// TIA Portal V20 export
// export: Created 2026-07-10T11:12:27.4069483Z, ExportSetting WithDefaults, DisplayName Totally Integrated Automation Portal, DisplayVersion V20, DisplayName TIA Portal Openness, DisplayVersion V20, DisplayName TIA Portal Version Control Interface, DisplayVersion V20, DisplayName STEP 7 Professional, DisplayVersion V20, DisplayName STEP 7 Safety, DisplayVersion V20, DisplayName WinCC Basic/Comfort/Advanced, DisplayVersion V20, DisplayName WinCC Unified, DisplayVersion V20
DATA_BLOCK "Inputs_DB"   // DB5
VERSION : 0.1
// stored: AutoNumber true, DBAccessibleFromOPCUA true, InstanceOfName Inputs, InstanceOfType FB
"Inputs"
   // VAR
   //    AIHandlers { S7_SetPoint := 'True'} : Array[0..5] of "AIHandler";
   //    WeightHandlers { S7_SetPoint := 'True'} : Array[0..1] of "WeightHandler";
   //    ErrorRCV1 { S7_SetPoint := 'True'} : Bool := TRUE;
   //    ErrorRCV2 { S7_SetPoint := 'True'} : Bool := TRUE;
   // END_VAR
BEGIN
   AIHandlers[0..3].Value := 32767.0;
   AIHandlers[4].Value := -13.0;
   AIHandlers[5].Value := 0.0;
   AIHandlers[0..3].ValueMin := 0.0;
   AIHandlers[4].ValueMin := 5320.0;
   AIHandlers[5].ValueMin := 0.0;
   AIHandlers[0..4].ValueMax := 27648.0;
   AIHandlers[5].ValueMax := 0.0;
   AIHandlers[0..5].ValueOffset := 0.0;
   AIHandlers[0..5].OutputMin := 0.0;
   AIHandlers[0..5].OutputMax := 0.0;
   AIHandlers[0..4].TimeBase := T#0MS;
   AIHandlers[5].TimeBase := T#1S;
   AIHandlers[0..4].Output := 0.0;
   AIHandlers[5].Output := 16#7FC0_0000;
   AIHandlers[0..5].Error := TRUE;
   AIHandlers[0..4].ConvertedValue := 0.0;
   AIHandlers[5].ConvertedValue := 16#7FC0_0000;
   AIHandlers[0..5].TON1.PT := T#2M;
   AIHandlers[0..5].TON1.IN := TRUE;
   AIHandlers[0..4].DelayTON.PT := T#0MS;
   AIHandlers[5].DelayTON.PT := T#20S;
   AIHandlers[0..4].DelayTON.IN := FALSE;
   AIHandlers[5].DelayTON.IN := TRUE;
   AIHandlers[0].FilterArray[0..199] := 0.0;
   AIHandlers[1].FilterArray[0..199] := 0.0;
   AIHandlers[2].FilterArray[0..199] := 0.0;
   AIHandlers[3].FilterArray[0..199] := 0.0;
   AIHandlers[4].FilterArray[0..199] := 0.0;
   AIHandlers[5].FilterArray[0..199] := 0.0;
   AIHandlers[0..4].FilterTime := T#0MS;
   AIHandlers[5].FilterTime := T#20S;
   AIHandlers[0..3].i := 17;
   AIHandlers[4].i := 28;
   AIHandlers[5].i := 29;
   AIHandlers[0..3].sum := 557039.0;
   AIHandlers[4].sum := -364.0;
   AIHandlers[5].sum := 0.0;
   AIHandlers[0..3].FilteredValue := 32767.0;
   AIHandlers[4].FilteredValue := -12.68;
   AIHandlers[5].FilteredValue := 0.0;
   AIHandlers[0..5].one := FALSE;
END_DATA_BLOCK
